FUNCTION_BLOCK FB_BiValve2Fdbck
VAR_INPUT
	mxReset						: BOOL;	(*Reset Error*)
	mxEmergency					: BOOL;
	mxAutoMode					: BOOL; (* TRUE = Automode *)
	mxCheckCilinder				: BOOL:= TRUE;
	mxIsVertical				: BOOL;
END_VAR
VAR_IN_OUT
	MachParameters					: ST_CilinderParameters;
END_VAR
VAR_OUTPUT
	mxIsIn						: BOOL;
	mxIsOut						: BOOL;
	mxIsOpen					: BOOL;
	mxIsClosed					: BOOL;
	Errors						: ST_CilinderErrors;
	
	mxErrorInit: BOOL;
	mxErrorStopInPos: BOOL;

END_VAR
VAR
	Check						: FB_CheckCilinder;
	
	QxIn	 					AT %Q*: BOOL;
	QxOut						AT %Q*: BOOL;
	IxIsIn						AT %I*: BOOL;
	IxIsOut						AT %I*: BOOL;

	mxHMI_In					: BOOL;
	mxHMI_Out					: BOOL;
	mxHMI_Open					: BOOL;
	mxHMI_Close					: BOOL;
	RT_HMI_In					: R_TRIG;
	RT_HMI_Out					: R_TRIG;
END_VAR

Error();

RT_HMI_In(CLK:= NOT mxAutoMode AND (mxHMI_In OR mxHMI_Open));
RT_HMI_Out(CLK:= NOT mxAutoMode AND (mxHMI_Out OR mxHMI_Close));

(* Manual *)
IF RT_HMI_In.Q THEN M_In(); END_IF
IF RT_HMI_Out.Q THEN M_Out(); END_IF

(* Reset Outputs *)

//IF IxIsIn THEN QxIn:= FALSE; END_IF
//IF IxIsOut THEN QxOut:= FALSE; END_IF

(* Status *)
mxIsIn:= mxIsOpen:= IxIsIn;
mxIsOut:= mxIsClosed:= IxIsOut;

ACTION Error:

IF NOT mxIsVertical THEN
	
	Check(
		MoveCilOut:= qxOut,
		MoveCilin:= qxIn,
		CheckCilinder:= mxCheckCilinder,
		SensorOut:=  mxIsOut OR mxIsClosed, // mx closed and open omgedraaid (20180528 -> Bateu*)
		SensorIn:= mxIsIn OR mxIsOpen,
		TimMax:= MachParameters.T_GuardTimeError,
		mxReset:= mxReset,
		ErrorCilinder=> Errors.Cilinder,
		ErrorCilinderOut=> ,
		ErrorCilinderIn=> ,
		ErrorEndNotReached=> ,
		ErrorSensorSwitched=> ,
		Time_Cil_Out=> ,
		Time_Cil_In=> );

(* Too slow errors, only messages *)

	Errors.CilinderSlow_IN	:=	mxCheckCilinder AND (Check.Time_Cil_In > MachParameters.T_GuardTimeWarning_IN);
	Errors.CilinderSlow_OUT	:=	mxCheckCilinder AND (Check.Time_Cil_Out > MachParameters.T_GuardTimeWarning_OUT);
END_IF

(**********************************************************************************************************)
mxErrorStopinPos:= FALSE;
mxErrorInit:= Errors.Cilinder;
END_ACTION

METHOD PUBLIC M_Close: BOOL
VAR_INPUT
END_VAR

IF NOT IxIsOut THEN QxOut:= TRUE; END_IF
QxIn:= FALSE;

(* Return value *)
M_Close:= IxIsOut;
END_METHOD

METHOD PUBLIC M_In : BOOL
VAR_INPUT
END_VAR

IF NOT IxIsIn THEN QxIn:= TRUE; END_IF
//QxIn:= TRUE;
QxOut:= FALSE;

(* Return value *)
M_In:= IxIsIn;
END_METHOD

METHOD PUBLIC M_In_Pressure : BOOL
VAR_INPUT
END_VAR
QxIn:= TRUE;
QxOut:= FALSE;

(* Return value *)
M_In_Pressure:= IxIsIn;
END_METHOD

METHOD PUBLIC M_Open : BOOL
VAR_INPUT
END_VAR

IF NOT IxIsIn THEN QxIn:= TRUE; END_IF
QxOut:= FALSE;

(* Return value *)
M_Open:= IxIsIn;
END_METHOD

METHOD PUBLIC M_Out: BOOL
VAR_INPUT
END_VAR

IF NOT IxIsOut THEN QxOut:= TRUE; END_IF
//qxOut:=TRUE;
QxIn:= FALSE;

(* Return value *)
M_Out:= IxIsOut;
END_METHOD

END_FUNCTION_BLOCK

(* stored: Version 1.1.0.1, ProductVersion 3.1.4020.12
   POU FB_BiValve2Fdbck: Id {b4b72d65-5a56-4ea4-96a5-faf3d225dd41}, SpecialFunc None
   Action Error: Id {b6861101-21e3-4269-ae3d-cc00c5b3378d}
   Method M_Close: Id {478a060a-3593-4b78-9ce1-84762883432e}
   Method M_In: Id {fa965505-a815-48c3-b9e1-76a49b9d8719}
   Method M_In_Pressure: Id {186dce28-0ba4-47c4-b075-e5d3483d54d5}
   Method M_Open: Id {63dc6af2-d7bd-48ce-b3fd-428d06b55477}
   Method M_Out: Id {1406251c-4949-40e6-9149-fd522861dd6b} *)
